FUNCTION_BLOCK FB_B EXTENDS FB_A
VAR_INPUT
    nVarB : INT := 0;
END_VAR

nVarA := 11;
nVarB := 2;

METHOD DoIt : BOOL
VAR_INPUT
END_VAR
VAR
    nVarB : INT;
END_VAR
nVarB := 22; // Se establece la variable local nVarB.
THIS^.nVarB := 222; // La variable del bloque de funciones nVarB se establece aunque nVarB está oculta.
F_FunA(fbMyFbA := THIS^);  //F_FunA es llamado via THIS^.
END_METHOD

END_FUNCTION_BLOCK

(* stored: Version 1.1.0.1, ProductVersion 3.1.4024.12
   POU FB_B: Id {e5dcf537-e5e1-4fcf-9687-be68b15b45a9}, SpecialFunc None
   Method DoIt: Id {ccefd84d-0001-4e09-91bc-d0ad1b59a78f} *)
